FUNCTION_BLOCK PUBLIC Load2Station
VAR_INPUT
END_VAR
VAR_OUTPUT
END_VAR
VAR
	xTrigger :BOOL := FALSE; // triggers processing
	State : eLoadSta2State := eLoadSta2State.eUnknown;
	NextState : eLoadSta2State := eLoadSta2State.eUnknown;
	bFirst : BOOL := TRUE;
	VUT : BYTE; //VehicleID Under Station
	DwellTimer : TON;
	LoadingComplete : BOOL := FALSE;
	CycleNumb: INT :=0;
	RowNumber :INT:=0;
	SeedNumber : INT:=9;
END_VAR

IF (GVL_IO.MachineEStopped) THEN 
	State := eLoadSta2State.eUnknown;
	NextState := eLoadSta2State.eUnknown;
END_IF

CASE State OF
eLoadSta2State.eUnknown:
	NextState := eLoadSta2State.eReady;

eLoadSta2State.eInit:

eLoadSta2State.eHoming:

eLoadSta2State.eReady:

   IF (xTrigger) THEN
		NextState := eLoadSta2State.eWaitForLoadComplete;
		
		DwellTimer(IN:=FALSE);		
	END_IF

eLoadSta2State.eDwell:

eLoadSta2State.eWaitForLoadComplete:
	 IF (LoadingComplete) THEN
		NextState := eLoadSta2State.eDepart;
        UpdatePartData();		
		LoadingComplete := FALSE;
		DwellTimer(IN:=FALSE);
	END_IF


eLoadSta2State.eProcessing:

eLoadSta2State.eDepart:
  	Stations.fbRoutePlanner.M_NotifyVehStaCmpl(StationIndex:= MM_CONST.LOAD_2_STA, VehicleID := VUT);
	xTrigger := FALSE;
	IF (Stations.fbCycleControl.StopRequested) THEN
		NextState := eLoadSta2State.eStopActive;
	ELSE	
		NextState := eLoadSta2State.eReady;	
	END_IF
	
eLoadSta2State.eStopActive:
	IF (NOT Stations.fbCycleControl.StopRequested) THEN
		NextState := eLoadSta2State.eReady;
	END_IF;
	
eLoadSta2State.eError:

END_CASE

IF (State <> NextState) THEN
	bFirst := TRUE;
ELSE
	bFirst := FALSE;
END_IF

State := NextState;
Status.StationsState[MM_CONST.LOAD_2_STA_HMI_STATE] := State;

METHOD PUBLIC ClearVehicleTrigger : BOOL
VAR_INPUT
END_VAR
xTrigger := FALSE;
END_METHOD

PROPERTY PUBLIC LoadComplete : BOOL
SET
LoadingComplete := LoadComplete;
END_SET
END_PROPERTY

METHOD PUBLIC ResetState : BOOL
VAR_INPUT
END_VAR
State := eLoadSta2State.eUnknown;
NextState := eLoadSta2State.eUnknown;
END_METHOD

METHOD PUBLIC SetRowNumber : BOOL
VAR_INPUT
	RowLocationNumber : INT;
END_VAR
RowNumber := RowLocationNumber;
END_METHOD

PROPERTY PUBLIC Trigger : BOOL
SET
xTrigger := Trigger;
END_SET
END_PROPERTY

METHOD PUBLIC UpdatePartData : BOOL
VAR_INPUT
END_VAR
memset(ADR(PartsData.Status[VUT]),0,SIZEOF(PartDataType));
PartsData.Status[VUT].LoadTime := SYSTEMTIME_TO_STRING(Logging.fbCurrTime.systemTime);
//PartsData.Status[VUT].CavityNumber := 5 + (CycleNumb MOD 4);
PartsData.Status[VUT].CavityNumber := RowNumber + SeedNumber;
CycleNumb := CycleNumb+1; // Use this till Yushin Robot sends out this information with Bit Location ID
PartsData.Status[VUT].OverallStatus := ePartStatus.eLoaded; // At least that is the assumption. We may want to check on how to turn off cavities later, but this will be caught by vision.
PartsData.Status[VUT].BarrelSize := LotsData.Lot.BarrelSize; // we are copying this data in case we might in future want to have more than one lots running at the same time on the machine
PartsData.Status[VUT].PartNumber := LotsData.Lot.PartNumber; // we are copying this data in case we might in future want to have more than one lots running at the same time on the machine
PartsData.Status[VUT].LotNumber := LotsData.Lot.LotNumber; // we are copying this data in case we might in future want to have more than one lots running at the same time on the machine
END_METHOD

PROPERTY PUBLIC VehicleUnderTest : BYTE
GET
VehicleUnderTest := VUT;
END_GET
SET
VUT := VehicleUnderTest;
END_SET
END_PROPERTY

END_FUNCTION_BLOCK

(* stored: Version 1.1.0.1, ProductVersion 3.1.4022.3
   POU Load2Station: Id {b3e7c2ce-ab66-48a1-9b42-5e93d26d4d56}, SpecialFunc None
   Method ClearVehicleTrigger: Id {9bccfcf9-f17f-4509-81b2-c06d4a7863c8}
   Property LoadComplete: Id {9331a946-1a99-446e-b80e-c3e9780d2d80}
   Set Set: Id {0af4b50f-5ae0-47e6-b5cd-67e3d6b518fc}
   Method ResetState: Id {10b2130d-ccad-459c-b83e-966aa985ab83}
   Method SetRowNumber: Id {7e43709c-36eb-4115-9f32-e43bdae1ce1c}
   Property Trigger: Id {bee5b29f-6b0b-4e6e-97fd-60a7cea0a2e4}
   Set Set: Id {8eb38652-2a0c-4492-be03-278a773fa17b}
   Method UpdatePartData: Id {46c8ff31-3bb6-4705-bd87-5ff346b87444}
   Property VehicleUnderTest: Id {6efe0dbf-6320-47f6-b295-7adbef2ce132}
   Get Get: Id {8c77a864-d3b5-4fcf-8308-3fefb1c6a88f}
   Set Set: Id {51f62ec0-bc16-4276-91a3-95d89569acc0} *)
